	REGION 7 - Prepare output data VFD

	    REGION 7.1 - Set speed setpoint in forward and reverse direction

	        #sR_TRIG_RunFWD(CLK := #iqUDT_ConveyorInterface.RunFwd);     // Get rising edge of Run forward signal
	        #sR_TRIG_RunRVS(CLK := #iqUDT_ConveyorInterface.RunRvs);     // Get rising edge of Run reverse signal

	        // When rising edge of the forward of reverse signal is received, the drive has to stop to be able to make the switch
	        IF #sR_TRIG_RunFWD.Q OR #sR_TRIG_RunRVS.Q
	        THEN
	            #qUDT_VfdOutputs.SetpointSpeed := 0;

	        END_IF;

	        // If motor stopped and Run forward is requested and forward direction is interlock, the speed setpoint is loaded to run forward.
	        IF (#iqUDT_ConveyorInterface.RunFwd) AND #iUDT_VfdConfig.InterlockFwd //(#i_UDT_VFDInputs.ActualSpeed = 0) AND
	        THEN
	            #sx_RunVfdForward := TRUE;
	            #sx_RunVfdReverse := FALSE;
	        END_IF;

	        // If motor stopped and Run reverse is requested and reverse direction is interlock, the speed setpoint is loaded to run forward.
	        IF (#iUDT_VfdInputs.ActualSpeed = 0) AND #iqUDT_ConveyorInterface.RunRvs AND #iUDT_VfdConfig.InterlockRvs
	        THEN
	            #sx_RunVfdReverse := TRUE;
	            #sx_RunVfdForward := FALSE;
	        END_IF;

	    END_REGION

	    REGION 7.2 - Stopping

	        // Create trigger when direction signal falling
	        #sF_TRIG_RunFwd(CLK := #iqUDT_ConveyorInterface.RunFwd);
	        #sF_TRIG_RunRvs(CLK := #iqUDT_ConveyorInterface.RunRvs);

	        // When no run signal or above run signal are given or drive is running and no occurs interlock (in specific direction) the VFD should stop
	        IF (NOT #iqUDT_ConveyorInterface.RunRvs AND NOT #iqUDT_ConveyorInterface.RunFwd)
	            OR (#iqUDT_ConveyorInterface.RunRvs AND #iqUDT_ConveyorInterface.RunFwd)
	            OR (#sx_RunVfdReverse AND NOT #iUDT_VfdConfig.InterlockRvs)
	            OR (#sx_RunVfdForward AND NOT #iUDT_VfdConfig.InterlockFwd)
	            OR #sF_TRIG_RunRvs.Q
	            OR #sF_TRIG_RunFwd.Q

	        THEN
	            #sx_RunVfdReverse := FALSE;
	            #sx_RunVfdForward := FALSE;
	        END_IF;

	        IF NOT #sx_RunVfdReverse AND NOT #sx_RunVfdForward AND (#iUDT_VfdInputs.ActualSpeed <> 0)
	        THEN
	            #sx_VfdStopping := TRUE;
	        ELSE
	            #sx_VfdStopping := FALSE;
	        END_IF;

	    END_REGION

	    REGION 7.3 - Check for enable operation signal

	        #sx_EnableOperation := #sx_VfdAvailable AND NOT #sx_ConfigurationError AND (#sx_RunVfdForward OR #sx_RunVfdReverse) OR #iqUDT_ConveyorInterface.VFDRunning;

	    END_REGION

	END_REGION

	REGION 8 - Write outputs to VFD

	    REGION 8.1 - Write control word 1

	        #qUDT_VfdOutputs.Control_Word_1.EnableRapidStop := #ix_QuickStopDisable;                       // Writing state to enable VFD to run
	        #qUDT_VfdOutputs.Control_Word_1.EnableApplicationStop := #sx_EnableOperation;                  // Writing state to Enable VFD operation
	        #qUDT_VfdOutputs.Control_Word_1.ReleaseBrake := FALSE;                                         // Not used
	        #qUDT_VfdOutputs.Control_Word_1.JogPos := FALSE;                                               // Not used
	        #qUDT_VfdOutputs.Control_Word_1.JogNeg := FALSE;                                               // Not used
	        #qUDT_VfdOutputs.Control_Word_1.ApplyRelativePositioning := FALSE;                             // Not used for speed control
	        #qUDT_VfdOutputs.Control_Word_1.StartStop := #sx_EnableOperation;                              // Writing state to start or stop VFD
	        #qUDT_VfdOutputs.Control_Word_1.ResetError := #iqUDT_ConveyorInterface.InternalErrorReset;    // Reseting VFD errors with error reset bit
	        #qUDT_VfdOutputs.Control_Word_1.ActivateDriveTrain2 := FALSE;                                  // Not used for MoviGear with one Drive Train
	        #qUDT_VfdOutputs.Control_Word_1.DeactivateSW_LimitSwitch := FALSE;                             // Not used
	        #qUDT_VfdOutputs.Control_Word_1.ActivateInhibit := NOT #sx_EnableOperation;                    // Controller Inhibit has TO be "false" before start/stop
	        #qUDT_VfdOutputs.Control_Word_1.ActivateStandby := FALSE;                                      // Not used
	        #qUDT_VfdOutputs.Control_Word_1.MovikitHandshakeIn := #sx_MovikitHandshakeIn;                  // MoviKit handshake controlled BY 0.5 Hz

	        // If hardware is unavailable clear the control word
	        IF NOT #sx_VfdAvailable
	        THEN
	            #qUDT_VfdOutputs.Control_Word_1.EnableRapidStop := FALSE;                                  // Writing state to enable VFD to run
	            #qUDT_VfdOutputs.Control_Word_1.EnableApplicationStop := FALSE;                            // Writing state to Enable VFD operation
	            #qUDT_VfdOutputs.Control_Word_1.ReleaseBrake := FALSE;                                     // Not used
	            #qUDT_VfdOutputs.Control_Word_1.JogPos := FALSE;                                           // Not used
	            #qUDT_VfdOutputs.Control_Word_1.JogNeg := FALSE;                                           // Not used
	            #qUDT_VfdOutputs.Control_Word_1.ApplyRelativePositioning := FALSE;                         // NOT used FOR speed control
	            #qUDT_VfdOutputs.Control_Word_1.StartStop := FALSE;                                        // Writing state to start or stop VFD
	            #qUDT_VfdOutputs.Control_Word_1.ResetError := FALSE;                                       // Reseting VFD errors with error reset bit
	            #qUDT_VfdOutputs.Control_Word_1.ActivateDriveTrain2 := FALSE;                              // Not used for MoviGear with one Drive Train
	            #qUDT_VfdOutputs.Control_Word_1.DeactivateSW_LimitSwitch := FALSE;                         // Not used
	            #qUDT_VfdOutputs.Control_Word_1.ActivateInhibit := FALSE;                                  // Controller Inhibit has TO be "false" before start/stop
	            #qUDT_VfdOutputs.Control_Word_1.ActivateStandby := FALSE;                                  // Not used
	            #qUDT_VfdOutputs.Control_Word_1.MovikitHandshakeIn := FALSE;                               // MoviKit handshake controlled BY 0.5 Hz
	            #qUDT_VfdOutputs.Control_Word_1.BIT_02_Reserved := FALSE;
	            #qUDT_VfdOutputs.Control_Word_1.BIT_09_Reserved := FALSE;
	            #qUDT_VfdOutputs.Control_Word_1.BIT_11_Reserved := FALSE;

	        END_IF;
	    END_REGION

	    REGION 8.2 - Write speed setpoint to drive
	        // The conveyor stopped and may now run in forward direction
	        IF (#sx_RunVfdForward AND NOT #iUDT_VfdConfig.DirectionReversal)
	            OR (#sx_RunVfdReverse AND #iUDT_VfdConfig.DirectionReversal)
	        THEN
	            #qUDT_VfdOutputs.SetpointSpeed := REAL_TO_INT(#sr_ActualSpeedSetpoint);
	        END_IF;

	        // The conveyor stopped and may now run in reverse direction
	        IF (#sx_RunVfdReverse AND NOT #iUDT_VfdConfig.DirectionReversal)
	            OR (#sx_RunVfdForward AND #iUDT_VfdConfig.DirectionReversal)

	        THEN
	            #qUDT_VfdOutputs.SetpointSpeed := REAL_TO_INT(#sr_ActualSpeedSetpoint * -1);
	        END_IF;

	        // Clear speed setpoint when no run request
	        IF NOT #sx_RunVfdForward AND NOT #sx_RunVfdReverse
	        THEN
	            #qUDT_VfdOutputs.SetpointSpeed := 0;
	        END_IF;

	    END_REGION

	    REGION 8.3 - Write acceleration and deceleration value to drive
	        // Write deceleration value to VFD
	        #qUDT_VfdOutputs.SetpointAcceleration := REAL_TO_INT(#iUDT_VfdConfig.ReferenceRPM / (UDINT_TO_REAL(#iUDT_VfdConfig.VFDRampUpTime) / 1000.0));        //Recalculating Acceleration ramp - deviding maximum configured speed by Ramp up time and devide it by 1000

	        // Write deceleration value to VFD
	        #qUDT_VfdOutputs.SetpointDeceleration := REAL_TO_INT(#iUDT_VfdConfig.ReferenceRPM / (UDINT_TO_REAL(#iUDT_VfdConfig.VFDRampDownTime) / 1000.0));      //Recalculating Deceleration ramp - deviding maximum configured speed by Ramp down time and devide it by 1000

	    END_REGION

	END_REGION

	REGION 9 - Check if motor is running

	    //The moto should start running after specific time. If nit the VFDRunningFeedback error occured
	    #sFB_TimerOnOffDelayVFDRunningFeedbackError(iudi_OnDelayTime := #iUDT_VfdConfig.VFDStartupTime,
	                                                ix_SignalToDelay := #sx_EnableOperation AND NOT (#si_ActualSpeed <> 0));

	    IF #sFB_TimerOnOffDelayVFDRunningFeedbackError.qx_DelayedSignal THEN

	        #sUDT_HMIStatus.VFDRunningFeedbackError := TRUE;

	    END_IF;

	END_REGION

	REGION 10 - Copy signals to interface DB and to status output UDT
	    // Create internal error status
	    #sx_ErrorActive := #sUDT_HMIStatus.PNSlaveNotonline
	    OR #sUDT_HMIStatus.PNSlaveError
	    OR #sUDT_HMIStatus.InternalError
	    OR #sUDT_HMIStatus.CommunicationErrorMovikit
	    OR #sUDT_HMIStatus.VFDRunningFeedbackError;

	    // Write interface bits
	    #iqUDT_ConveyorInterface.VFDRunning := #iUDT_VfdInputs.Status_Word_1.DriveActive AND #sx_VfdAvailable AND #iqUDT_ConveyorInterface.ActualSpeed <> 0;        // Write true on output Conveyor interface structure if VFD is in operation and motor is turning
	    #iqUDT_ConveyorInterface.VFDatSpeed := #sx_SpeedSetpointReached AND #sx_VfdAvailable;                                                                         // Copy setpoint speed reached state from static  to the output conveyor interface structure
	    #iqUDT_ConveyorInterface.InternalWarningVFD := #iUDT_VfdInputs.Status_Word_1.Warning;                                                                         // Set the internal VFD warning bit if any warning is active
	    #iqUDT_ConveyorInterface.InternalErrorVFD := #sx_ErrorActive;                                                                                                  // Set the internal VFD error bit if any fault is active
	    #iqUDT_ConveyorInterface.ActualSpeed := #si_ActualSpeed;                                                                                                       // Copy the calculated value to the output
	    #iqUDT_ConveyorInterface.ConfigurationError := #iqUDT_ConveyorInterface.ConfigurationError OR #sx_ConfigurationError;

	    // Copy error status to output
	    #qUDT_HMIStatus := #sUDT_HMIStatus;
	END_REGION

	REGION 11 - Statistics
	    // Create trigger on error and create statistics for profinet slave not online
	    #sR_TRIG_PNSlaveNotOnline(CLK := #sUDT_HMIStatus.PNSlaveNotonline);                              // Detect the rising edge of the error

	    IF #iqUDT_ConveyorInterface.ResetStatistics OR #sUDT_HMIStatus.PNSlaveNotonline
	    THEN

	        "FC_Statistics"(ix_Reset := #iqUDT_ConveyorInterface.ResetStatistics,
	                        ix_Activate := #sUDT_HMIStatus.PNSlaveNotonline,
	                        ix_RTrigActivate := #sR_TRIG_PNSlaveNotOnline.Q,
	                        iqUDT_Statistics := #iqUDT_VfdStatistics.PNSlaveNotOnline);
	    END_IF;

	    // Create trigger on error and create statistics for profinet slave error
	    #sR_TRIG_PNSlaveError(CLK := #sUDT_HMIStatus.PNSlaveError);                                      // Detect the rising edge of the error

	    IF #iqUDT_ConveyorInterface.ResetStatistics OR #sUDT_HMIStatus.PNSlaveError
	    THEN

	        "FC_Statistics"(ix_Reset := #iqUDT_ConveyorInterface.ResetStatistics,
	                        ix_Activate := #sUDT_HMIStatus.PNSlaveError,
	                        ix_RTrigActivate := #sR_TRIG_PNSlaveError.Q,
	                        iqUDT_Statistics := #iqUDT_VfdStatistics.PNSlaveError);
	    END_IF;

	    // Create trigger on error and create statistics for internal VFD Error
	    #sR_TRIG_InternalError(CLK := #sUDT_HMIStatus.InternalError);                                    // Detect the rising edge of the error

	    IF #iqUDT_ConveyorInterface.ResetStatistics OR #sUDT_HMIStatus.InternalError
	    THEN

	        "FC_Statistics"(ix_Reset := #iqUDT_ConveyorInterface.ResetStatistics,
	                        ix_Activate := #sUDT_HMIStatus.InternalError,
	                        ix_RTrigActivate := #sR_TRIG_InternalError.Q,
	                        iqUDT_Statistics := #iqUDT_VfdStatistics.VFDInternalError);
	    END_IF;

	    // Create trigger on error and create statistics for Movikit communication error
	    #sR_TRIG_CommunicationErrorMovikit(CLK := #sUDT_HMIStatus.CommunicationErrorMovikit);            // Detect the rising edge of the error

	    IF #iqUDT_ConveyorInterface.ResetStatistics OR #sUDT_HMIStatus.CommunicationErrorMovikit
	    THEN

	        "FC_Statistics"(ix_Reset := #iqUDT_ConveyorInterface.ResetStatistics,
	                        ix_Activate := #sUDT_HMIStatus.CommunicationErrorMovikit,
	                        ix_RTrigActivate := #sR_TRIG_CommunicationErrorMovikit.Q,
	                        iqUDT_Statistics := #iqUDT_VfdStatistics.CommunicationErrorMovikit);
	    END_IF;

	    // Create trigger on running signal and create statistics for running status
	    #sR_TRIG_Running(CLK := #iqUDT_ConveyorInterface.VFDRunning);                                 // Detect the rising edge of the signal

	    IF #iqUDT_ConveyorInterface.ResetStatistics OR #iqUDT_ConveyorInterface.VFDRunning
	    THEN

	        "FC_Statistics"(ix_Reset := #iqUDT_ConveyorInterface.ResetStatistics,
	                        ix_Activate := #iqUDT_ConveyorInterface.VFDRunning,
	                        ix_RTrigActivate := #sR_TRIG_Running.Q,
	                        iqUDT_Statistics := #iqUDT_VfdStatistics.Running);
	    END_IF;
	END_REGION

	REGION 12 - VFD codes
	    (*
	    FCB number |                       | Meaning
	    ______________________________________________________________________________________________________________
	        1                               Output stage inhibit
	        2                               Default stop
	        4                               Manual Mode
	        5                               Speed control
	                101                     Speed-controlled jogging. Encoder feedback NOT required.
	                200                     Speed control. Encoder feedback NOT required.
	        6                               Interpolated speed control
	        7                               Torque control
	        8                               Interpolated torque control
	        9                               Positioning mode
	                400                     Absolute position control
	                401                     Relative position control
	                402                     Modulo position control - positive
	                403                     Modulo position control - negative
	                404                     Modulo position control - shortest distance
	        10                              Interpolated position control
	        12                              Referencing mode
	                300                     Reference travel - offset via parameter
	                301                     Reference travel - offset via fieldbus
	        13                              Stop at application limits
	        14                              Emergency stop
	        18                              Rotor position identification
	        19                              Position hold control
	        20                              Jog mode
	                100                     Position-controlled jogging. Encoder feedback required
	        21                              Brake test
	        25                              Motor parameter measurement
	        26                              Stop at user limits

	    Error code | Suberror code        | Meaning                                | Measure
	    ______________________________________________________________________________________________________________
	        3       1                       Ground fault                            Consult "Fault table" in
	        4       1                       Brake chopper fault                     document 'SEW Movigear-C 25887130.PDF'
	        6       1                       Line fault                              Chapter 8.7
	        7       1                       DC link fault
	        8       1,2,3                   Speed monitoring fault
	        9       1,2,5,6,9,10            Control mode fault
	        10      1,3-11                  Data flexibility fault
	        11      1-6                     Temperature monitoring fault
	        12      1,2                     Fault brake
	        13      5,24                    Encoder 1 fault
	        16      5-8,10,20-27            Startup fault
	        19      1-9                     Process data fault
	        20      2,11                    Fault device monitoring
	        23      4                       Power section fault
	        25      2-7,20,21,30,31,61,70   Parameter memory monitoring
	        26      1,3                     External fault
	        28      1-12,14                 FCB drive function fault
	        29      1-4                     Hardware limit switch fault
	        30      1-3                     Software limit switch fault
	        31      1-4,7,9                 Thermal protection fault
	        32      2-6,12                  Communication fault
	        33      11,12,13                system initialisation fault
	        34      1                       Process data configuration fault
	        35      1-5                     Function activation fault
	        42      1-3                     Lag fault
	        46      2,3,50,51,52            Safety card fault
	        51      1                       Analog processing fault

	    Error code | Suberror code        | Meaning                                | Measure
	    ______________________________________________________________________________________________________________
	        1       1,2                     Output stage monitoring fault           Contact SEW-Eurodrive Service
	        4       2                       Brake chopper fault
	        7       2                       DC link fault
	        9       3,4,8                   Control mode fault
	        10      2,99                    Data flexibility fault
	        11      7,8                     Temperature monitoring fault
	        13      1,3,6,7.8,9,11,13,      Encoder 1 fault
	                15,22,23
	        16      2,11,12,30              Startup fault
	        17      7                       Internal processor fault
	        18      1,3,4,7,8,9,10,12,13    Software fault
	        20      1,7                     Fault device monitoring
	        21      1                       S-Drive 1 fault
	        23      5,6,7,8                 Power section fault
	        25      10,12-19,50,51,81       Parameter memory monitoring
	        28      13                      FCB drive funcyio fault
	        33      1,2,6,7,8,10            System initialisation fault
	        46      1                       Safety card fault

	    Function Control Block (FCB) codes
	    FBC = 01 Output stage inhibit
	    FBC = 02 Default stop
	    FBC = 04 Manual Mode
	    FBC = 05 Speed control
	     101 - Speed-controlled jogging. Encoder feedback NOT required.
	     200 - Speed control. Encoder feedback NOT required.
	    FBC = 06 Interpolated speed control
	    FBC = 07 Torque control
	    FBC = 08 Interpolated torque control
	    FBC = 09 Positioning mode
	    400 - Absolute position control
	    401 - Relative position control
	    402 - Modulo position control - positive
	    403 - Modulo position control - negative
	    404 - Modulo position control - shortest distance
	    FBC = 10 Interpolated position control
	    FBC = 12 Referencing mode
	    300 - Reference travel - offset via parameter
	    301 - Reference travel - offset via fieldbus
	    FBC = 13 Stop at application limits
	    FBC = 14 Emergency stop
	    FBC = 18 Rotor position identification
	    FBC = 19 Position hold control
	    FBC = 20 Jog mode
	     100 - Position-controlled jogging. Encoder feedback required
	    FBC = 21 Brake test
	    FBC = 25 Motor parameter measurement
	    FBC = 26 Stop at user limits

	    *)
	END_REGION
END_FUNCTION_BLOCK

FUNCTION_BLOCK "FB_VfdSEWMOVI-CPositioning"
TITLE = FB_VFD_SEW_MOVI-C_Positioning
{ S7_Optimized_Access := 'TRUE' }
AUTHOR : MHSE
VERSION : 3.0
// ATTRIBUTES
// AUTO_NUMBER = True
// BLOCK_NUMBER = 36
// END_ATTRIBUTES
//Control SEW Servo VFD with multiple positions
   VAR_INPUT
      iUDT_VfdConfig { ExternalAccessible := 'False'; ExternalVisible := 'False'; ExternalWritable := 'False'} : "UDT_VfdPositioningConfiguration";   //  Configuration structure
      iUDT_VfdInputs { ExternalAccessible := 'False'; ExternalVisible := 'False'; ExternalWritable := 'False'} : "UDT_VfdSEWPositioningPI";   //  VFD inputs structure
      ix_MainPowerOk { ExternalAccessible := 'False'; ExternalVisible := 'False'; ExternalWritable := 'False'} : Bool;   //  True = Main power is ok
      ix_BackupPowerOk { ExternalAccessible := 'False'; ExternalVisible := 'False'; ExternalWritable := 'False'} : Bool;   //  True = back-up power is ok
      ix_SimulationModeActive { ExternalAccessible := 'False'; ExternalVisible := 'False'; ExternalWritable := 'False'} : Bool;   //  Simulation On
   END_VAR

   VAR_OUTPUT
      qUDT_HMIStatus { ExternalAccessible := 'False'; ExternalVisible := 'False'; ExternalWritable := 'False'} : "UDT_VfdPositioningStatus";   //  HMI status structure
      qUDT_VfdOutputs { ExternalAccessible := 'False'; ExternalVisible := 'False'; ExternalWritable := 'False'} : "UDT_VfdSEWPositioningPO";   //  VFD outputs structure
   END_VAR

   VAR_IN_OUT
      iqUDT_VSUInterface : "UDT_VSUInterface";   //  VSU interface structure
      iqUDT_VFDStatistics : "UDT_VfdStatistics";   //  VFD statistics
   END_VAR

   VAR
      sUDT_PNDevice { ExternalAccessible := 'False'; ExternalVisible := 'False'; ExternalWritable := 'False'; S7_SetPoint := 'False'} : "UDT_PNDevice";   //  PN device info structure
      sUDT_HMIStatus { ExternalAccessible := 'False'; ExternalVisible := 'False'; ExternalWritable := 'False'; S7_SetPoint := 'False'} : "UDT_VfdPositioningStatus";   //  Status struture
      sFB_TimerOnOffDelayCheckSupply { ExternalAccessible := 'False'; ExternalVisible := 'False'; ExternalWritable := 'False'; S7_SetPoint := 'False'} : "FB_TimerOnOffDelay";   //  MHS "TimerOnOffDelay" - to delay time for VFD supply contactor
      sFB_TimerOnOffDelayMoviKit { ExternalAccessible := 'False'; ExternalVisible := 'False'; ExternalWritable := 'False'; S7_SetPoint := 'False'} : "FB_TimerOnOffDelay";   //  MHS "TimerOnOffDelay" - to delay time for MoviKit response delay error
      sFB_TimerOnOffDelayPositioning { ExternalAccessible := 'False'; ExternalVisible := 'False'; ExternalWritable := 'False'; S7_SetPoint := 'False'} : "FB_TimerOnOffDelay";   //  MHS "TimerOnOffDelay" - to delay time for Porisioning delay error
      sFB_TimerOnOffDelayFasterManualSpeed { ExternalAccessible := 'False'; ExternalVisible := 'False'; ExternalWritable := 'False'; S7_SetPoint := 'False'} : "FB_TimerOnOffDelay";
      sFB_TimerOnOffDelayActivateInhibit { ExternalAccessible := 'False'; ExternalVisible := 'False'; ExternalWritable := 'False'; S7_SetPoint := 'False'} : "FB_TimerOnOffDelay";
      sF_TRIG_LST {InstructionName := 'F_TRIG'; LibVersion := '1.0'; ExternalAccessible := 'False'; ExternalVisible := 'False'; ExternalWritable := 'False'; S7_SetPoint := 'False'} : F_TRIG;   //  Falling edge positioning feedback
      sR_TRIG_ManInPos {InstructionName := 'R_TRIG'; LibVersion := '1.0'; ExternalAccessible := 'False'; ExternalVisible := 'False'; ExternalWritable := 'False'; S7_SetPoint := 'False'} : R_TRIG;   //  Rising edge manual travel into position
      sR_TRIG_PNSlaveNotOnline {InstructionName := 'R_TRIG'; LibVersion := '1.0'; ExternalAccessible := 'False'; ExternalVisible := 'False'; ExternalWritable := 'False'; S7_SetPoint := 'False'} : R_TRIG;   //  Rising edge for trigger Profinet slave not online statistics
      sR_TRIG_PNSlaveError {InstructionName := 'R_TRIG'; LibVersion := '1.0'; ExternalAccessible := 'False'; ExternalVisible := 'False'; ExternalWritable := 'False'; S7_SetPoint := 'False'} : R_TRIG;   //  Rising edge for trigger Profinet slave error statistics
      sR_TRIG_InternalError {InstructionName := 'R_TRIG'; LibVersion := '1.0'; ExternalAccessible := 'False'; ExternalVisible := 'False'; ExternalWritable := 'False'; S7_SetPoint := 'False'} : R_TRIG;   //  Rising edge for trigger Internal VFD Error statistics
      sR_TRIG_CommunicationErrorMovikit {InstructionName := 'R_TRIG'; LibVersion := '1.0'; ExternalAccessible := 'False'; ExternalVisible := 'False'; ExternalWritable := 'False'; S7_SetPoint := 'False'} : R_TRIG;   //  Rising edge for trigger communication error Movikit statistics
      sR_TRIG_Running {InstructionName := 'R_TRIG'; LibVersion := '1.0'; ExternalAccessible := 'False'; ExternalVisible := 'False'; ExternalWritable := 'False'; S7_SetPoint := 'False'} : R_TRIG;   //  Rising edge for starting of the running signal
      sa_PNPortsStatus { ExternalAccessible := 'False'; ExternalVisible := 'False'; ExternalWritable := 'False'} : Array[1..8] of Bool;   // TRUE when specific port has an error
      sr_ActualTorque { ExternalAccessible := 'False'; ExternalVisible := 'False'; ExternalWritable := 'False'} : Real;   //  Actual torque of drive
      sdi_ActualPositionValue { ExternalAccessible := 'False'; ExternalVisible := 'False'; ExternalWritable := 'False'} : DInt;   //  Actual position in mm
      si_ManualSpeed { ExternalAccessible := 'False'; ExternalVisible := 'False'; ExternalWritable := 'False'} : Int;   //  Actual manual speed
      si_ActualSpeed { ExternalAccessible := 'False'; ExternalVisible := 'False'; ExternalWritable := 'False'} : Int;   //  Actual speed in mm/s
      si_LastSwitchtime { ExternalAccessible := 'False'; ExternalVisible := 'False'; ExternalWritable := 'False'} : Int;   //  The actual time it took the last switch-over
      sx_ErrorActive { ExternalAccessible := 'False'; ExternalVisible := 'False'; ExternalWritable := 'False'} : Bool;   //  An error is active
      sx_WarningActive { ExternalAccessible := 'False'; ExternalVisible := 'False'; ExternalWritable := 'False'} : Bool;   //  A warning is active
      sx_PNDeviceHealthy { ExternalAccessible := 'False'; ExternalVisible := 'False'; ExternalWritable := 'False'} : Bool;   //  PN Device is healthy, no errors
      sx_MovikitHandshakeIn { ExternalAccessible := 'False'; ExternalVisible := 'False'; ExternalWritable := 'False'} : Bool;   //  Handshake to movikit
      sx_MoviKitFeedback { ExternalAccessible := 'False'; ExternalVisible := 'False'; ExternalWritable := 'False'} : Bool;   //  Movikit feedback delay
      sx_HardwareAvailable { ExternalAccessible := 'False'; ExternalVisible := 'False'; ExternalWritable := 'False'} : Bool;   //  All hardware is on line and available
      sx_PowerOK { ExternalAccessible := 'False'; ExternalVisible := 'False'; ExternalWritable := 'False'} : Bool;   //  All Power (in and external) is ok
      sx_PositioningFeedback { ExternalAccessible := 'False'; ExternalVisible := 'False'; ExternalWritable := 'False'} : Bool;   //  Positioning feedback delay
      sx_VFDReady { ExternalAccessible := 'False'; ExternalVisible := 'False'; ExternalWritable := 'False'} : Bool;   //  The VFD control is ready to operate
      sx_StartVFD { ExternalAccessible := 'False'; ExternalVisible := 'False'; ExternalWritable := 'False'} : Bool;   //  Start VFD
      sx_MotorRunning { ExternalAccessible := 'False'; ExternalVisible := 'False'; ExternalWritable := 'False'} : Bool;   //  The servo motor is running
      sx_ManualPositionStop { ExternalAccessible := 'False'; ExternalVisible := 'False'; ExternalWritable := 'False'} : Bool;   //  A configured position is reached in manual mode
      sx_ManualPosHold { ExternalAccessible := 'False'; ExternalVisible := 'False'; ExternalWritable := 'False'} : Bool;   //  Hold in position
      sx_RestartMan { ExternalAccessible := 'False'; ExternalVisible := 'False'; ExternalWritable := 'False'} : Bool;   //  Manual restart requested
      sx_ConfigurationError { ExternalAccessible := 'False'; ExternalVisible := 'False'; ExternalWritable := 'False'} : Bool;   //  Commissioning: configuration of parameters is wrong
      si_LoopCounter { ExternalAccessible := 'False'; ExternalVisible := 'False'; ExternalWritable := 'False'} : Int;
      sx_Check { ExternalAccessible := 'False'; ExternalVisible := 'False'; ExternalWritable := 'False'} : Bool;
   END_VAR

   VAR_TEMP
      tdi_EncoderPositionSetpoint : DInt;   //  Value of position setpoint
   END_VAR

   VAR CONSTANT
      ci_NumberOfProfinetPorts : Int := 2;   // Number of Profinet ports in device
      ci_SpeedManualMode : Int := 100;   // Speed in manual mode for jogging
      ci_SpeedManualModeAfter5s : Int := 200;
   END_VAR


BEGIN
	(*
	----------------------------------------------------------------------------------------

	Version history:
	Date        | Version   | Author        | Remark
	----------------------------------------------------------------------------------------
	24/05/2019  | 0.1       | P. Majka      | first release MHS TIA 15.1
	29/07/2019  | 0.2       | P. Majka      | Adding new functionality - comments to change
	30/07/2019  | 2.0       | P. Majka      | Moved to project with library 2.0
	31/07/2019  | 2.1       | M. Kurpiers   | Updating comments
	08/08/2019  | 2.2       | J.Krawczuk    | Updating referencing
	14/08/2019  | 2.3       | J.Krawczuk    | Added new functionality
	24/08/2019  | 2.4       | F. Baten      | Changed regions / combined errors / modified comments and working
	05/11/2019  | 2.5       | S.Theocharis  | Change the VFDDeviceName to VFDPNDeviceName for consistency with rest VFD blocks
	20/11/2019  | 2.10      | S. Nikodem    | Configuration error
	20/11/2019  | 3.0       | P.Majka       | 3.0 MHS library release TIA 15.1
	28/02/2020  | 3.1       | F.Baten       | Reinstated positioning warning (Servo takes too long to get to position) and
	                                        | separated it again from OutOfPosition error (over running the set positions)
	01/02/2020  | 3.2       | F.Baten       | Changed "UDT_VFD_Status" to "UDT_VFD_PositioningStatus"
	04/02/2020  | 3.3       | F.Baten       | Changed VSU Rio interface - Error and ready modified.
	06/08/2020  | 3.4       | L.Klar        | Manual speed changed
	03/11/2020  | 3.5       | K.Pokorski    | Profinet ports diagnostics added
	21/02/2023  | 4.0       | F.Baten       | 4.0 Release TIA 17.5
	06/10/2023  | 4.1       | F.Baten       | All positions converted to DINT as need of higher values for lift funtion
	14/06/2024  | 4.1       | R.Pieczonka   | Changed conditions for "EnableApplicationStop". Fixed setting output speed
	*)

	REGION 1 - Get Device Profinet information

	    "FC_GetDevicePN"(is_PNDeviceName := #iUDT_VfdConfig.VFDPNDeviceName,
	                     ix_SimulationModeActive := #ix_SimulationModeActive,
	                     iqUDT_PND := #sUDT_PNDevice);


	    "FC_GetPNPortStatus"(ii_NumberOfPorts := #ci_NumberOfProfinetPorts,
	                         iUDT_DevicePNInfo := #sUDT_PNDevice,
	                         qa_PortFault => #sa_PNPortsStatus);

	END_REGION

	REGION 2 - Reset errors

	    IF #iqUDT_VSUInterface.InternalErrorReset

	    THEN
	        #sUDT_HMIStatus.CommunicationErrorMovikit := FALSE;                    // The Movikit application is not reacting
	        #sUDT_HMIStatus.PNSlaveNotOnline := FALSE;                             // Profinet slave is not on line
	        #sUDT_HMIStatus.PNSlaveError := FALSE;                                 // Profinet slave has an error
	        #sUDT_HMIStatus.PositioningTimeOutError := FALSE;                      // Reset positioning error
	        #sUDT_HMIStatus.InternalError := FALSE;                                // Reset internal error
	        #sUDT_HMIStatus.PNSlaveWarning := FALSE;


	    END_IF;

	END_REGION

	REGION 3 - Check Hardware

	    REGION 3.1 - Power OK
	        // Hardware will be available after delay so the device has time for initialisation
	        #sFB_TimerOnOffDelayCheckSupply(iudi_OnDelayTime := 2000,              // Set time for on delay
	                                        ix_SignalToDelay := #ix_MainPowerOk);  // Mains are ok

	        #sx_PowerOK := #sFB_TimerOnOffDelayCheckSupply.qx_DelayedSignal;       // And All Power (in and external) is ok
	    END_REGION

	    REGION 3.2 - PN Healthy Check

	        IF NOT "DB_ProfinetDiagnostic".ProfinetNetworks[#sUDT_PNDevice.PNNetworknumber].DeviceStatus[#sUDT_PNDevice.PNDeviceNumber].DeviceState.Exist     // Or the connected device doesn't exist
	            AND NOT #ix_SimulationModeActive                                    // And not in simulation
	            AND (#sx_PowerOK                                                    // Main Power is ok
	            OR #ix_BackupPowerOk)                                               // Or backup power is ok
	        THEN
	            #sUDT_HMIStatus.PNSlaveNotOnline := TRUE;
	        END_IF;

	        // Check if PN ports are healthy
	        IF #sa_PNPortsStatus[1] XOR #sa_PNPortsStatus[2] THEN
	            #sUDT_HMIStatus.PNSlaveWarning := TRUE;
	        END_IF;

	        IF "DB_ProfinetDiagnostic".ProfinetNetworks[#sUDT_PNDevice.PNNetworknumber].DeviceStatus[#sUDT_PNDevice.PNDeviceNumber].DeviceState.Error       // Or the device has an error
	            AND NOT #ix_SimulationModeActive                                    // And not in simulation
	            AND (#sx_PowerOK                                                    // Main Power is ok
	            OR #ix_BackupPowerOk)                                               // Or backup power is ok
	            AND NOT #sUDT_HMIStatus.PNSlaveWarning                             // and PN ports are healthy

	        THEN
	            #sUDT_HMIStatus.PNSlaveError := TRUE;                              // Profinet slave has an error
	        END_IF;

	        #sx_PNDeviceHealthy := NOT #sUDT_HMIStatus.PNSlaveNotOnline            // Or the device an error
	        AND NOT #sUDT_HMIStatus.PNSlaveError                                   // Profinet slave has an error
	        AND (#sx_PowerOK                                                        // Main Power is ok
	        OR #ix_BackupPowerOk)                                                   // Or backup power is ok
	        AND #sUDT_PNDevice.PNDeviceFound;                                      // Device is found in network configuration

	    END_REGION

	    // Hardware is available
	    #sx_HardwareAvailable := #iUDT_VfdInputs.Status_Word_1.STO_Inactive        // Safety is ok
	    AND #sx_PowerOK                                                             // All mains are ok
	    AND #sx_PNDeviceHealthy                                                     // No PN errors
	    OR #ix_SimulationModeActive;                                                // Or simulation active

	    REGION 3.3 - Check communication MoviKit
	        #sx_MoviKitFeedback :=                                                  // Set MoviKit feedback delay
	        ((#sx_MovikitHandshakeIn                                                // IF MoviKit handshake input is active
	        AND NOT #iUDT_VfdInputs.Status_Word_1.MovikitHandshakeOut)             // And MoviKit handshake output active
	        OR (NOT #sx_MovikitHandshakeIn                                          // Or MoviKit handshake input isn't active
	        AND #iUDT_VfdInputs.Status_Word_1.MovikitHandshakeOut));               // And MoviKit handshake output isn't active

	        #sFB_TimerOnOffDelayMoviKit(iudi_OnDelayTime := 1000,                  // Set on delay time to 1000
	                                    ix_SignalToDelay := NOT #sx_MoviKitFeedback);          // Start timer

	        IF (#sFB_TimerOnOffDelayMoviKit.qx_DelayedSignal)                      // If the timer elapsed
	            AND #sx_HardwareAvailable
	        THEN
	            #sUDT_HMIStatus.CommunicationErrorMovikit := TRUE;                 // Set MoviKit error
	        END_IF;

	        #sx_MovikitHandshakeIn := NOT #iUDT_VfdInputs.Status_Word_1.MovikitHandshakeOut;   // Set the Handshake signal
	    END_REGION


	END_REGION

	REGION 4 - Handle input data

	    REGION 4.1 - Move to status

	        #sr_ActualTorque := INT_TO_REAL(#iUDT_VfdInputs.ActualTorque) / 1000.0 * #iUDT_VfdConfig.TorqueMax;   // Writing actual real calculated torque
	        #si_ActualSpeed := #iUDT_VfdInputs.ActualSpeed;                                                        // Actual speed in mm/s
	        #sx_MotorRunning := #iUDT_VfdInputs.Status_Word_1.DriveActive;                                         // Set status motor running if motor shaft is turning

	    END_REGION

	    REGION 4.2 - Actual positon value

	        #sdi_ActualPositionValue := SHL(IN := (WORD_TO_DINT(IN := #iUDT_VfdInputs.ActualPosition_hW)), N := 16) + WORD_TO_DINT(IN := #iUDT_VfdInputs.ActualPosition_lW);   // Calculate actual encoder position from two words

	        IF #sdi_ActualPositionValue <= (#iUDT_VfdConfig.Position[#iqUDT_VSUInterface.PositionSetpoint] + #iUDT_VfdConfig.PositionWindow)         // If actual encoder position in mm is lower or equal to position setpoint plus position window
	            AND #sdi_ActualPositionValue >= (#iUDT_VfdConfig.Position[#iqUDT_VSUInterface.PositionSetpoint] - #iUDT_VfdConfig.PositionWindow)    // And actual encoder position in mm is greater or equal to position setpoint minus position window

	        THEN
	            #iqUDT_VSUInterface.PositionActual := #iqUDT_VSUInterface.PositionSetpoint;                                              // Write position setpoint TO actual position number when position setpoint reached
	        ELSIF #iqUDT_VSUInterface.Manual
	        THEN
	            #sx_Check := FALSE;
	            FOR #si_LoopCounter := 0 TO "FC_GetNrOfArrayEl"(iv_Array := #iUDT_VfdConfig.Position) DO
	                IF #sdi_ActualPositionValue <= (#iUDT_VfdConfig.Position[#si_LoopCounter] + #iUDT_VfdConfig.PositionWindow)
	                    AND #sdi_ActualPositionValue >= (#iUDT_VfdConfig.Position[#si_LoopCounter] - #iUDT_VfdConfig.PositionWindow)
	                THEN
	                    #iqUDT_VSUInterface.PositionActual := #si_LoopCounter;
	                    #sx_Check := TRUE;
	                END_IF;
	            END_FOR;
	            IF #sx_Check = 0 THEN
	                #iqUDT_VSUInterface.PositionActual := 0;
	            END_IF;
	        ELSE
	            #iqUDT_VSUInterface.PositionActual := 0;
	        END_IF;




	    END_REGION

	    REGION 4.3 - Manual position
	        // to stop at a predefined position when jogging, after the stop the movement can continue by pressing the jogbutton again
	        IF #iUDT_VfdInputs.Mode = 100                                                                          // The actual application mode is equal to 100
	        THEN
	            #sx_ManualPositionStop :=
	            (#sdi_ActualPositionValue <= (#iUDT_VfdConfig.Position[1] + #iUDT_VfdConfig.PositionWindow)       // IF actual encoder position in mm is lower OR equal TO position setpoint plus position window
	            AND #sdi_ActualPositionValue >= (#iUDT_VfdConfig.Position[1] - #iUDT_VfdConfig.PositionWindow))   // And actual encoder position in mm is greater or equal to position setpoint minus position window
	            OR (#sdi_ActualPositionValue <= (#iUDT_VfdConfig.Position[2] + #iUDT_VfdConfig.PositionWindow)    // IF actual encoder position in mm is lower OR equal TO position setpoint plus position window
	            AND #sdi_ActualPositionValue >= (#iUDT_VfdConfig.Position[2] - #iUDT_VfdConfig.PositionWindow))   // And actual encoder position in mm is greater or equal to position setpoint minus position window
	            OR (#sdi_ActualPositionValue <= (#iUDT_VfdConfig.Position[3] + #iUDT_VfdConfig.PositionWindow)    // IF actual encoder position in mm is lower OR equal TO position setpoint plus position window
	            AND #sdi_ActualPositionValue >= (#iUDT_VfdConfig.Position[3] - #iUDT_VfdConfig.PositionWindow))   // And actual encoder position in mm is greater or equal to position setpoint minus position window
	            OR (#sdi_ActualPositionValue <= (#iUDT_VfdConfig.Position[4] + #iUDT_VfdConfig.PositionWindow)    // IF actual encoder position in mm is lower OR equal TO position setpoint plus position window
	            AND #sdi_ActualPositionValue >= (#iUDT_VfdConfig.Position[4] - #iUDT_VfdConfig.PositionWindow))   // And actual encoder position in mm is greater or equal to position setpoint minus position window
	            OR (#sdi_ActualPositionValue <= (#iUDT_VfdConfig.Position[5] + #iUDT_VfdConfig.PositionWindow)    // IF actual encoder position in mm is lower OR equal TO position setpoint plus position window
	            AND #sdi_ActualPositionValue >= (#iUDT_VfdConfig.Position[5] - #iUDT_VfdConfig.PositionWindow))   // And actual encoder position in mm is greater or equal to position setpoint minus position window
	            OR (#sdi_ActualPositionValue <= (#iUDT_VfdConfig.Position[6] + #iUDT_VfdConfig.PositionWindow)    // IF actual encoder position in mm is lower OR equal TO position setpoint plus position window
	            AND #sdi_ActualPositionValue >= (#iUDT_VfdConfig.Position[6] - #iUDT_VfdConfig.PositionWindow))   // And actual encoder position in mm is greater or equal to position setpoint minus position window
	            OR (#sdi_ActualPositionValue <= (#iUDT_VfdConfig.Position[7] + #iUDT_VfdConfig.PositionWindow)    // IF actual encoder position in mm is lower OR equal TO position setpoint plus position window
	            AND #sdi_ActualPositionValue >= (#iUDT_VfdConfig.Position[7] - #iUDT_VfdConfig.PositionWindow))   // And actual encoder position in mm is greater or equal to position setpoint minus position window
	            OR (#sdi_ActualPositionValue <= (#iUDT_VfdConfig.Position[8] + #iUDT_VfdConfig.PositionWindow)    // IF actual encoder position in mm is lower OR equal TO position setpoint plus position window
	            AND #sdi_ActualPositionValue >= (#iUDT_VfdConfig.Position[8] - #iUDT_VfdConfig.PositionWindow))   // And actual encoder position in mm is greater or equal to position setpoint minus position window
	            OR (#sdi_ActualPositionValue <= (#iUDT_VfdConfig.Position[9] + #iUDT_VfdConfig.PositionWindow)    // IF actual encoder position in mm is lower OR equal TO position setpoint plus position window
	            AND #sdi_ActualPositionValue >= (#iUDT_VfdConfig.Position[9] - #iUDT_VfdConfig.PositionWindow))   // And actual encoder position in mm is greater or equal to position setpoint minus position window
	            OR (#sdi_ActualPositionValue <= (#iUDT_VfdConfig.Position[10] + #iUDT_VfdConfig.PositionWindow)   // IF actual encoder position in mm is lower OR equal TO position setpoint plus position window
	            AND #sdi_ActualPositionValue >= (#iUDT_VfdConfig.Position[10] - #iUDT_VfdConfig.PositionWindow)); // And actual encoder position in mm is greater or equal to position setpoint minus position window
	        END_IF;
	    END_REGION
	END_REGION

	REGION 5 - Errors and warnings

	    REGION 5.1 - VFD internal error

	        #sUDT_HMIStatus.InternalError := #iUDT_VfdInputs.Status_Word_1.Error; // An internal VFD error is active
	        #sUDT_HMIStatus.ErrorCode := #iUDT_VfdInputs.StatusErrorNo.%B1;       // Copy VFD error code from static status structure to HMI status structure
	        #sUDT_HMIStatus.SubErrorCode := #iUDT_VfdInputs.StatusErrorNo.%B0;    // Copy VFD sub-error code from static status structure to HMI status structure

	        IF NOT #iUDT_VfdInputs.Status_Word_1.Error
	            AND NOT #iUDT_VfdInputs.Status_Word_1.Warning
	        THEN
	            #sUDT_HMIStatus.ErrorCode := 0;                                    // Copy VFD error code from static status structure TO HMI status structure
	            #sUDT_HMIStatus.SubErrorCode := 0;                                 // Copy VFD sub-error code from static status structure to HMI status structure
	        END_IF;
	    END_REGION

	    REGION 5.2 - Positioning error
	        // This timer checks if the speed of the VFD is ok.
	        // The VFD should reach is next destination in the given time
	        //

	        #sx_PositioningFeedback := #iqUDT_VSUInterface.PositionActual <> #iqUDT_VSUInterface.PositionSetpoint // If actual position is different than setpoint position
	        AND #iqUDT_VSUInterface.Automatic;                                                                     // And in automatic mode

	        #sF_TRIG_LST(CLK := #sx_PositioningFeedback);

	        IF #sF_TRIG_LST.Q
	        THEN
	            #si_LastSwitchtime := LREAL_TO_INT(#sFB_TimerOnOffDelayPositioning.qlr_ActualTime);
	        END_IF;



	        #sFB_TimerOnOffDelayPositioning(iudi_OnDelayTime := (#iqUDT_VSUInterface.SwitchingTime),  // Set on delay time
	                                        ix_SignalToDelay := #sx_PositioningFeedback);              // Start timer when positioning feedback delay



	        IF #sFB_TimerOnOffDelayPositioning.qx_DelayedSignal                    // If the time elapsed
	        THEN

	            #sUDT_HMIStatus.PositioningTimeOutError := TRUE;                   // Set positioning warning

	        END_IF;
	    END_REGION

	    REGION 5.3 - Common Error
	        // Set VFD error active
	        #sx_ErrorActive := #sUDT_HMIStatus.InternalError                       // The VFD indicates an active error
	        OR #sUDT_HMIStatus.CommunicationErrorMovikit;                          // The block generated an communication error

	    END_REGION

	    REGION 5.4 - Configuration Warning
	        //  Check if no faulty setup is active
	        //  This is the responcebility of the commisioning engineer

	        IF #iUDT_VfdConfig.PositionMax > #iUDT_VfdConfig.PositionMin          // Max position is bigger than min position
	            AND #iUDT_VfdConfig.PositionMax > 0                                // and not 0
	            AND #iUDT_VfdConfig.VFDSpeed > 0                                   // Max speed is not 0
	            AND #iUDT_VfdConfig.VFDAccDecel > 0                                // Maximum acceleration an deceleration time is not 0
	            AND "DB_ProfinetDiagnostic".ProfinetNetworks[#sUDT_PNDevice.PNNetworknumber].DeviceStatus[#sUDT_PNDevice.PNDeviceNumber].DeviceState.Configure
	        THEN
	            #sx_ConfigurationError := FALSE;                                    // Reset the configuration warning
	        ELSE
	            #sx_ConfigurationError := TRUE;                                     // Set configuration warning
	        END_IF;
	    END_REGION

	    REGION 5.5 - Common warning
	        // Set VFD warning active
	        #sx_WarningActive := #iUDT_VfdInputs.Status_Word_1.Warning             // The VFD indicates an active warning
	        OR #sUDT_HMIStatus.PositioningTimeOutError;                                 // The VFD did not reach the position in time.

	    END_REGION

	END_REGION

	REGION 6 - Check conditions to set VFD Ready signals

	    REGION 6.1 - Internal VFD ready

	        #sx_VFDReady := #sx_HardwareAvailable                                   // The hardware is powered up and detected
	        AND (#iUDT_VfdInputs.Status_Word_1.InverterReady                       // And VFD is ready to start
	        OR #sx_MotorRunning)                                                    // Or motor running
	        AND NOT #sx_ErrorActive                                                 // And no VFD error active
	        AND NOT #sx_ConfigurationError;
	        // AND NOT (#iqUDT_VSUInterface.PositionActual = #iqUDT_VSUInterface.RequestedPosition);    /// Commented out because  it was causing issues for the refernce drive                                // And no configuration error

	    END_REGION

	    REGION 6.2 - External VFD ready (to control)

	        #iqUDT_VSUInterface.Ready :=                                           // Signal ready is active if:
	        (#iqUDT_VSUInterface.Automatic                                         // And automatic mode request
	        AND NOT #iqUDT_VSUInterface.Manual                                     // And no manual mode request
	        AND #iUDT_VfdInputs.Status_Word_1.Referenced                           // And the drive is referenced
	        AND #iUDT_VfdInputs.Mode = 400)                                        // Actual application mode is equal to 400
	        OR
	        (NOT #iqUDT_VSUInterface.Automatic                                     // No automatic mode request
	        AND #iqUDT_VSUInterface.Manual                                         // AND manual mode request
	        AND #iUDT_VfdInputs.Mode = 100)                                        // And the actual application mode is equal to 100
	        OR
	        (#iqUDT_VSUInterface.Reference_command                                 // And the "refference" command is active
	        AND #iUDT_VfdInputs.Mode = 301)                                        // The actual application mode is equal TO 301
	        AND
	        (#sx_VFDReady                                                           // Status ready is active
	        AND #iqUDT_VSUInterface.RunEnabled);                                   // And running of the lifting device is enabled by VSU

	    END_REGION
	END_REGION

	REGION 7 - Set VFD control data

	    REGION 7.1 - Stop VFD

	        IF NOT #iqUDT_VSUInterface.Ready                                       // If VFD isn't ready to operate
	        THEN

	            #sx_StartVFD := FALSE;                                              // Reset start VFD
	            #qUDT_VfdOutputs.SetpointMode := 0;                                // Set the application mode to 0

	        END_IF;

	    END_REGION

	    REGION 7.3 - Reference VFD

	        IF #sx_VFDReady                                                         // If status VFD ready to operate is active
	            AND #iqUDT_VSUInterface.Reference_command                          // And the "refference" command is active
	        THEN

	            #qUDT_VfdOutputs.SetpointMode := 301;                              // Selecting FCB for reference travel FCB = 12

	            #tdi_EncoderPositionSetpoint := #iUDT_VfdConfig.Position[0];                                  // Set the position value as refference
	            #qUDT_VfdOutputs.SetpointPosition_hW := DINT_TO_WORD(SHR(IN := (#tdi_EncoderPositionSetpoint), N := 16));  // Send new position to encoder - high word
	            #qUDT_VfdOutputs.SetpointPosition_lW := DINT_TO_WORD(IN := #tdi_EncoderPositionSetpoint);                  // Send new position TO encoder - low word
	        END_IF;


	        IF #iqUDT_VSUInterface.Ready AND                                       // If VFD system is ready to operation
	            #iUDT_VfdInputs.Mode = 301                                         // And actual application mode  is equal to 301
	        THEN

	            #sx_StartVFD := TRUE;                                               // Set start VFD

	        END_IF;

	    END_REGION

	    REGION 7.4 - Manual mode - jogging

	        IF #sx_VFDReady                                                         // If status VFD ready to operation is active
	            AND #iqUDT_VSUInterface.Manual                                     // And manual mode request is active
	            AND NOT #iqUDT_VSUInterface.Automatic                              // And automatic mode request isn't active
	            AND #iqUDT_VSUInterface.RunEnabled                                 // And running of the lifting device is enabled by VSU
	            AND NOT #iqUDT_VSUInterface.Reference_command                      // And the "refference" command isn't active

	        THEN

	            #qUDT_VfdOutputs.SetpointMode := 100;                              // Selecting FCB for position-controlled jogging FCB = 20

	        END_IF;

	        // On position while jogging: stop, when button is released and pressed again continue to travel
	        //
	        #sR_TRIG_ManInPos(CLK := #sx_ManualPositionStop);

	        #sx_ManualPosHold := (#sx_ManualPosHold                                 // Hold movement as long as buttons are pressed
	        OR #sR_TRIG_ManInPos.Q)                                                // trigger position reached
	        AND (#iqUDT_VSUInterface.JogUp                                         // jogging up active
	        OR #iqUDT_VSUInterface.JogDown)                                        // jogging down active
	        AND #iqUDT_VSUInterface.Ready;                                         // ready to operate

	        // Jog commands

	        IF #iqUDT_VSUInterface.Ready                                           // If the VFD system is ready to operate
	            AND (#iUDT_VfdInputs.Mode = 100)                                   // And the actual application mode is equal to 100
	            AND #iqUDT_VSUInterface.JogUp                                      // And selected jog in positive direction
	            AND NOT #iqUDT_VSUInterface.JogDown                                // And not selected jog in negative direction
	            AND NOT #sx_ManualPosHold
	        THEN

	            #qUDT_VfdOutputs.Control_Word_1.JogPos := TRUE;                                                // Set jog positive VFD control bit
	            #qUDT_VfdOutputs.Control_Word_1.JogNeg := FALSE;                                               // Reset jog negative VFD control bit

	        ELSIF
	            #iqUDT_VSUInterface.Ready                                          // If the VFD system is ready to operate
	            AND (#iUDT_VfdInputs.Mode = 100)                                   // And the actual application mode is equal to 100
	            AND NOT #iqUDT_VSUInterface.JogUp                                  // And not selected jog in positive direction
	            AND #iqUDT_VSUInterface.JogDown                                    // And selected jog in negative direction
	            AND NOT #sx_ManualPosHold
	        THEN

	            #qUDT_VfdOutputs.Control_Word_1.JogPos := FALSE;                   // Reset jog positive VFD control bit
	            #qUDT_VfdOutputs.Control_Word_1.JogNeg := TRUE;                    // Set jog negative VFD control bit

	        ELSE

	            #qUDT_VfdOutputs.Control_Word_1.JogPos := FALSE;                   // Reset jog positive VFD control bit
	            #qUDT_VfdOutputs.Control_Word_1.JogNeg := FALSE;                   // Reset jog negative VFD control bit

	        END_IF;

	    END_REGION

	    REGION 7.5 - Automatic mode - for positioning

	        IF #sx_VFDReady                                                         // If status VFD ready to operation is active
	            AND #iqUDT_VSUInterface.Automatic                                  // And automatic mode request is active
	            AND NOT #iqUDT_VSUInterface.Manual                                 // And manual mode request isn't active
	            AND #iqUDT_VSUInterface.RunEnabled                                 // And running of the lifting device is enabled by VSU
	            AND #iUDT_VfdInputs.Status_Word_1.Referenced                       // And the drive is referenced
	            AND NOT #iqUDT_VSUInterface.Reference_command                      // And the "refference" command isn't active

	        THEN

	            #qUDT_VfdOutputs.SetpointMode := 400;                              // Select FCB for absolute positioning control FCB = 09

	        END_IF;

	        IF #iqUDT_VSUInterface.Ready AND                                       // IF VFD system is ready TO operation
	            #iUDT_VfdInputs.Mode = 400                                         // And actual application mode is equal to 400
	        THEN

	            #tdi_EncoderPositionSetpoint := #iUDT_VfdConfig.Position[#iqUDT_VSUInterface.PositionSetpoint];    // Move position request to setpoint postion
	            #qUDT_VfdOutputs.SetpointPosition_hW := DINT_TO_WORD(SHR(IN := (#tdi_EncoderPositionSetpoint), N := 16));         // Send new position to encoder - high word
	            #qUDT_VfdOutputs.SetpointPosition_lW := DINT_TO_WORD(IN := #tdi_EncoderPositionSetpoint);                         // Send new position to encoder - low word
	            #sx_StartVFD := TRUE;

	        END_IF;

	    END_REGION


	    REGION 7.6 - Set output speed

	        // When the drive was manual operated, first start in manual speed to go to position

	        #si_ManualSpeed := #ci_SpeedManualMode;                                 // Manual speed setpoint

	        IF (#iqUDT_VSUInterface.Manual                                          // Manual command is activated
	            OR #iqUDT_VSUInterface.GoReference)
	            AND NOT #iqUDT_VSUInterface.Automatic
	        THEN
	            #sx_RestartMan := TRUE;                                             // Set memory Manual was activated
	        END_IF;

	        IF #iqUDT_VSUInterface.PositionActual = #iqUDT_VSUInterface.PositionSetpoint     // Signal from VFD, indicating being in position
	            OR #iqUDT_VSUInterface.Automatic
	        THEN
	            #sx_RestartMan := FALSE;                                            // Reset memory Manual was activated
	        END_IF;


	        IF #iUDT_VfdInputs.Mode = 400                                          // If actual application mode is Auto ( 400 )
	        THEN
	            IF NOT #sx_RestartMan                                               // Manual was not activated

	            THEN
	                #qUDT_VfdOutputs.SetpointSpeed := #iUDT_VfdConfig.VFDSpeed;   // Move speedsetpoint to output
	            ELSE                                                                // If manual was activated then
	                #qUDT_VfdOutputs.SetpointSpeed := #si_ManualSpeed;             // Move manual speedsetpoint to output
	            END_IF;

	        ELSIF #iUDT_VfdInputs.Mode = 100                                       // If actual application mode is manual ( 100 )
	        THEN

	            #qUDT_VfdOutputs.SetpointSpeed := #si_ManualSpeed;                 // Move manual speedsetpoint TO output

	        END_IF;

	    END_REGION


	    REGION 7.8 - Other control signals to VFD

	        #qUDT_VfdOutputs.Control_Word_1.EnableRapidStop := (#sx_HardwareAvailable AND #iqUDT_VSUInterface.RunEnabled); // Writing states of VFD power is ready or simulation to enable VFD to run
	        #qUDT_VfdOutputs.Control_Word_1.EnableApplicationStop := #sx_VFDReady AND ((NOT (#sdi_ActualPositionValue = #tdi_EncoderPositionSetpoint) AND #iqUDT_VSUInterface.Automatic) OR (#iqUDT_VSUInterface.Manual AND ((#iqUDT_VSUInterface.JogDown OR #iqUDT_VSUInterface.JogUp) OR #iqUDT_VSUInterface.Reference_command)));                             // Writing state to enable VFD operation
	        #qUDT_VfdOutputs.Control_Word_1.ReleaseBrake := FALSE;                                             // Not used
	        #qUDT_VfdOutputs.Control_Word_1.ApplyRelativePositioning := FALSE;                                 // Not used for speed control
	        #qUDT_VfdOutputs.Control_Word_1.StartStop := #sx_StartVFD;                                         // Writing state to start or stop VFD
	        #qUDT_VfdOutputs.Control_Word_1.ResetError := #iqUDT_VSUInterface.InternalErrorReset;             // Reseting VFD errors with error reset bit
	        #qUDT_VfdOutputs.Control_Word_1.ActivateDriveTrain2 := FALSE;                                      // Not used for MoviGear with on Drive Train
	        #qUDT_VfdOutputs.Control_Word_1.DeactivateSW_LimitSwitch := FALSE;                                 // Not used
	        #qUDT_VfdOutputs.Control_Word_1.ActivateInhibit := NOT #sx_VFDReady;                                // Controller Inhibit has to be "false" before start/stop
	        #qUDT_VfdOutputs.Control_Word_1.ActivateStandby := FALSE;                                          // Not used
	        #qUDT_VfdOutputs.Control_Word_1.MovikitHandshakeIn := #sx_MovikitHandshakeIn;                      // Set "MoviKit" handshake input to 1 by 0.5 sec.

	    END_REGION

	    REGION 7.9 - Acceleration and deceleration ramps

	        #qUDT_VfdOutputs.SetpointAcceleration := #iUDT_VfdConfig.VFDAccDecel;
	        #qUDT_VfdOutputs.SetpointDeceleration := #iUDT_VfdConfig.VFDAccDecel;

	    END_REGION

	END_REGION

	REGION 8 - In case of communication error reset VFD outputs

	    IF NOT #sx_HardwareAvailable                                                                            // If hardware is not available

	    THEN

	        #qUDT_VfdOutputs.Control_Word_1.ResetError := FALSE;                                               // Reset reset VFD error
	        #qUDT_VfdOutputs.Control_Word_1.ActivateDriveTrain2 := FALSE;                                      // Reset activate drive train
	        #qUDT_VfdOutputs.Control_Word_1.DeactivateSW_LimitSwitch := FALSE;                                 // Reset deactivate software limit switch
	        #qUDT_VfdOutputs.Control_Word_1.ActivateInhibit := FALSE;                                          // Reset activate inhibit
	        #qUDT_VfdOutputs.Control_Word_1.ActivateStandby := FALSE;                                          // Reset activate standby
	        #qUDT_VfdOutputs.Control_Word_1.MovikitHandshakeIn := FALSE;                                       // Reset movikit hanshake input
	        #qUDT_VfdOutputs.Control_Word_1.EnableRapidStop := FALSE;                                          // Reset enable rapid stop
	        #qUDT_VfdOutputs.Control_Word_1.EnableApplicationStop := FALSE;                                    // Reset enable application stop
	        #qUDT_VfdOutputs.Control_Word_1.ReleaseBrake := FALSE;                                             // Reset release brake
	        #qUDT_VfdOutputs.Control_Word_1.JogPos := FALSE;                                                   // Reset jog in positive direction
	        #qUDT_VfdOutputs.Control_Word_1.JogNeg := FALSE;                                                   // Reset jog in negative direction
	        #qUDT_VfdOutputs.Control_Word_1.ApplyRelativePositioning := FALSE;                                 // Reset applying relatice positioning
	        #qUDT_VfdOutputs.Control_Word_1.StartStop := FALSE;                                                // Reset Start/Stop VFD
	    END_IF;
	END_REGION

	REGION 9 - Statistics

	    // Number OF times the VFD had an internal error

	    #sR_TRIG_PNSlaveNotOnline(CLK := #sUDT_HMIStatus.PNSlaveNotOnline);       // Detect the rising edge of the error

	    IF #iqUDT_VSUInterface.ResetStatistics OR                                  // If there is signal to reset statistics from VSU interface
	        #sUDT_HMIStatus.PNSlaveNotOnline                                       // Or the error occured
	    THEN

	        "FC_Statistics"(ix_Reset := #iqUDT_VSUInterface.ResetStatistics,       // Reset statistics
	                        ix_Activate := #sUDT_HMIStatus.PNSlaveNotOnline,       // Actual error
	                        ix_RTrigActivate := #sR_TRIG_PNSlaveNotOnline.Q,       // Trigger rising edge error
	                        iqUDT_Statistics := #iqUDT_VFDStatistics.PNSlaveNotOnline);   // Statistics structure
	    END_IF;

	    // Number of ethernet communication faults to VFD drive

	    #sR_TRIG_PNSlaveError(CLK := #sUDT_HMIStatus.PNSlaveError);               // Detect the rising edge of the error
	    IF #iqUDT_VSUInterface.ResetStatistics OR                                  // If there is signal to reset statistics from VSU interface
	        #sUDT_HMIStatus.PNSlaveError                                           // Or the error occured
	    THEN

	        "FC_Statistics"(ix_Reset := #iqUDT_VSUInterface.ResetStatistics,       // Reset statistics
	                        ix_Activate := #sUDT_HMIStatus.PNSlaveError,           // Actual error
	                        ix_RTrigActivate := #sR_TRIG_PNSlaveError.Q,           // Trigger rising edge error
	                        iqUDT_Statistics := #iqUDT_VFDStatistics.PNSlaveError);       // Statistics structure

	    END_IF;


	    // Number of times the VFD had an internal error

	    #sR_TRIG_InternalError(CLK := #sUDT_HMIStatus.InternalError);             // Detect the rising edge of the error

	    IF #iqUDT_VSUInterface.ResetStatistics OR                                  // IF there is signal TO reset statistics from VSU interface
	        #sUDT_HMIStatus.InternalError                                          // Or the error occured
	    THEN

	        "FC_Statistics"(ix_Reset := #iqUDT_VSUInterface.ResetStatistics,       // Reset statistics
	                        ix_Activate := #sUDT_HMIStatus.InternalError,          // Actual error
	                        ix_RTrigActivate := #sR_TRIG_InternalError.Q,          // Trigger rising edge error
	                        iqUDT_Statistics := #iqUDT_VFDStatistics.VFDInternalError);       // Statistics structure

	    END_IF;

	    // Number OF times the VFD had a safety error

	    #sR_TRIG_CommunicationErrorMovikit(CLK := #sUDT_HMIStatus.CommunicationErrorMovikit); // Detect the rising edge of the error

	    IF #iqUDT_VSUInterface.ResetStatistics OR                                  // If there is signal to reset statistics from VSU interface
	        #sUDT_HMIStatus.CommunicationErrorMovikit                              // Or the error occured
	    THEN

	        "FC_Statistics"(ix_Reset := #iqUDT_VSUInterface.ResetStatistics,       // Reset statistics
	                        ix_Activate := #sUDT_HMIStatus.CommunicationErrorMovikit,              // Actual error
	                        ix_RTrigActivate := #sR_TRIG_CommunicationErrorMovikit.Q,              // Trigger rising edge error
	                        iqUDT_Statistics := #iqUDT_VFDStatistics.CommunicationErrorMovikit);  // Statistics structure

	    END_IF;

	    // Number of times the VFD has been running

	    #sR_TRIG_Running(CLK := #iUDT_VfdInputs.Status_Word_1.DriveActive);       // Detect the rising edge of the signal

	    IF #iqUDT_VSUInterface.ResetStatistics OR                                  // If there is signal to reset statistics from VSU interface
	        #iUDT_VfdInputs.Status_Word_1.STO_Inactive                             // Or the status occured
	    THEN

	        "FC_Statistics"(ix_Reset := #iqUDT_VSUInterface.ResetStatistics,       // Reset statistics
	                        ix_Activate := #iUDT_VfdInputs.Status_Word_1.DriveActive,  // Actual status
	                        ix_RTrigActivate := #sR_TRIG_Running.Q,                // Trigger rising edge
	                        iqUDT_Statistics := #iqUDT_VFDStatistics.Running);    // Statistics structure

	    END_IF;
	END_REGION

	REGION 10 - Write interface outputs

	    //Internal Error
	    #iqUDT_VSUInterface.InternalErrorVFD := #sx_ErrorActive;                   // Set the internal VFD error bit in VSU interface IF Any fault is active

	    //Internal Warning
	    #iqUDT_VSUInterface.InternalWarningVFD := #sx_WarningActive;               // Set the internal VFD warning bit if any warning is active

	    //Motor running
	    #iqUDT_VSUInterface.MotorRunning := #iUDT_VfdInputs.Status_Word_1.DriveActive;    // Set motor is running in VSU interface IF status control Word "motor running" is active

	    //Send signal VFD is referenced
	    #iqUDT_VSUInterface.Referenced := #iUDT_VfdInputs.Status_Word_1.Referenced;       // Write state of drive is referenced from VFD to VSU interface


	    #iqUDT_VSUInterface.Positioning := #iqUDT_VSUInterface.PositionSetpoint <> #iqUDT_VSUInterface.PositionActual  // Set the lifting device is positioning if position setpoint is different than actual position
	    AND #iqUDT_VSUInterface.Automatic                                      // AND automatic mode enabled
	    AND NOT #iqUDT_VSUInterface.InternalErrorVFD;                          // And internal error VFD no occurred

	    #iqUDT_VSUInterface.StartLowSpeed := #sx_RestartMan;                       // Indicating to VSU the VSD is starting in low speed

	    #qUDT_HMIStatus := #sUDT_HMIStatus;                                       // Copy status to output
	END_REGION

	REGION 11 - error codes
	    (*
	    FCB number |                       | Meaning
	    ______________________________________________________________________________________________________________
	        1                               Output stage inhibit
	        2                               Default stop
	        4                               Manual Mode
	        5                               Speed control
	                101                     Speed-controlled jogging. Encoder feedback NOT required.
	                200                     Speed control. Encoder feedback NOT required.
	        6                               Interpolated speed control
	        7                               Torque control
	        8                               Interpolated torque control
	        9                               Positioning mode
	                400                     Absolute position control
	                401                     Relative position control
	                402                     Modulo position control - positive
	                403                     Modulo position control - negative
	                404                     Modulo position control - shortest distance
	        10                              Interpolated position control
	        12                              Referencing mode
	                300                     Reference travel - offset via parameter
	                301                     Reference travel - offset via fieldbus
	        13                              Stop at application limits
	        14                              Emergency stop
	        18                              Rotor position identification
	        19                              Position hold control
	        20                              Jog mode
	                100                     Position-controlled jogging. Encoder feedback required
	        21                              Brake test
	        25                              Motor parameter measurement
	        26                              Stop at user limits


	    Error code | Suberror code        | Meaning                                | Measure
	    ______________________________________________________________________________________________________________
	        3       1                       Ground fault                            Consult "Fault table" in
	        4       1                       Brake chopper fault                     document 'SEW Movigear-C 25887130.PDF'
	        6       1                       Line fault                              Chapter 8.7
	        7       1                       DC link fault
	        8       1,2,3                   Speed monitoring fault
	        9       1,2,5,6,9,10            Control mode fault
	        10      1,3-11                  Data flexibility fault
	        11      1-6                     Temperature monitoring fault
	        12      1,2                     Fault brake
	        13      5,24                    Encoder 1 fault
	        16      5-8,10,20-27            Startup fault
	        19      1-9                     Process data fault
	        20      2,11                    Fault device monitoring
	        23      4                       Power section fault
	        25      2-7,20,21,30,31,61,70   Parameter memory monitoring
	        26      1,3                     External fault
	        28      1-12,14                 FCB drive function fault
	        29      1-4                     Hardware limit switch fault
	        30      1-3                     Software limit switch fault
	        31      1-4,7,9                 Thermal protection fault
	        32      2-6,12                  Communication fault
	        33      11,12,13                system initialisation fault
	        34      1                       Process data configuration fault
	        35      1-5                     Function activation fault
	        42      1-3                     Lag fault
	        46      2,3,50,51,52            Safety card fault
	        51      1                       Analog processing fault

	    Error code | Suberror code        | Meaning                                | Measure
	    ______________________________________________________________________________________________________________
	        1       1,2                     Output stage monitoring fault           Contact SEW-Eurodrive Service
	        4       2                       Brake chopper fault
	        7       2                       DC link fault
	        9       3,4,8                   Control mode fault
	        10      2,99                    Data flexibility fault
	        11      7,8                     Temperature monitoring fault
	        13      1,3,6,7.8,9,11,13,      Encoder 1 fault
	                15,22,23
	        16      2,11,12,30              Startup fault
	        17      7                       Internal processor fault
	        18      1,3,4,7,8,9,10,12,13    Software fault
	        20      1,7                     Fault device monitoring
	        21      1                       S-Drive 1 fault
	        23      5,6,7,8                 Power section fault
	        25      10,12-19,50,51,81       Parameter memory monitoring
	        28      13                      FCB drive funcyio fault
	        33      1,2,6,7,8,10            System initialisation fault
	        46      1                       Safety card fault

	    Function Control Block (FCB) codes
	    FBC = 01 Output stage inhibit
	    FBC = 02 Default stop
	    FBC = 04 Manual Mode
	    FBC = 05 Speed control
	     101 - Speed-controlled jogging. Encoder feedback NOT required.
	     200 - Speed control. Encoder feedback NOT required.
	    FBC = 06 Interpolated speed control
	    FBC = 07 Torque control
	    FBC = 08 Interpolated torque control
	    FBC = 09 Positioning mode
	    400 - Absolute position control
	    401 - Relative position control
	    402 - Modulo position control - positive
	    403 - Modulo position control - negative
	    404 - Modulo position control - shortest distance
	    FBC = 10 Interpolated position control
	    FBC = 12 Referencing mode
	    300 - Reference travel - offset via parameter
	    301 - Reference travel - offset via fieldbus
	    FBC = 13 Stop at application limits
	    FBC = 14 Emergency stop
	    FBC = 18 Rotor position identification
	    FBC = 19 Position hold control
	    FBC = 20 Jog mode
	     100 - Position-controlled jogging. Encoder feedback required
	    FBC = 21 Brake test
	    FBC = 25 Motor parameter measurement
	    FBC = 26 Stop at user limits

	    *)
	END_REGION
END_FUNCTION_BLOCK

FUNCTION_BLOCK "FB_RIOVSU"
TITLE = FB_RIOVSU
{ S7_Optimized_Access := 'TRUE' }
AUTHOR : MHSE
FAMILY : GeneralSystemFunctions
VERSION : 3.0
// ATTRIBUTES
// AUTO_NUMBER = True
// BLOCK_NUMBER = 226
// END_ATTRIBUTES
   VAR_INPUT
      is_ET200spPNDeviceName { ExternalAccessible := 'False'; ExternalVisible := 'False'; ExternalWritable := 'False'} : String;   //   Name of the ET200sp device
      ix_400VintOk { ExternalAccessible := 'False'; ExternalVisible := 'False'; ExternalWritable := 'False'} : Bool;   //   TRUE if internal circuit breaker 400V is ok
      ix_400VextOk { ExternalAccessible := 'False'; ExternalVisible := 'False'; ExternalWritable := 'False'} : Bool;   //   TRUE if external 400V Main cabinet is ok
      ix_BrakeSupplyOk { ExternalAccessible := 'False'; ExternalVisible := 'False'; ExternalWritable := 'False'} : Bool;   //   TRUE if circuit breaker of brake power supply is ok
      ix_ThermalBrake { ExternalAccessible := 'False'; ExternalVisible := 'False'; ExternalWritable := 'False'} : Bool;   //   TRUE when No thermal error
      ix_24VOk { ExternalAccessible := 'False'; ExternalVisible := 'False'; ExternalWritable := 'False'} : Bool;   //   TRUE when 24V power supply to RIO is ok
      ix_SimulationModeActive { ExternalAccessible := 'False'; ExternalVisible := 'False'; ExternalWritable := 'False'} : Bool;   //   True when Simulation mode active
      ix_HardwareOk { ExternalAccessible := 'False'; ExternalVisible := 'False'; ExternalWritable := 'False'} : Bool;   //  TRUE when  hardware is Ok
   END_VAR

   VAR_OUTPUT
      qUDT_HMIStatus { ExternalAccessible := 'False'; ExternalVisible := 'False'; ExternalWritable := 'False'} : "UDT_RIOVSUStatus";   //   HMI status structure
   END_VAR

   VAR_IN_OUT
      iqUDT_Statistics : "UDT_RIOVSUStatistics";   //   Statistics structure
      iqUDT_VSUInterface : "UDT_VSUInterface";   //   Interface RIO and VSU
   END_VAR

   VAR
      sUDT_HMIStatus { ExternalAccessible := 'False'; ExternalVisible := 'False'; ExternalWritable := 'False'; S7_SetPoint := 'False'} : "UDT_RIOVSUStatus";   //   HMI status structure
      sUDT_PNDevice { ExternalAccessible := 'False'; ExternalVisible := 'False'; ExternalWritable := 'False'; S7_SetPoint := 'False'} : "UDT_PNDevice";   //   PN device structure
      sa_PNPortsStatus { ExternalAccessible := 'False'; ExternalVisible := 'False'; ExternalWritable := 'False'} : Array[1..8] of Bool;   // TRUE when specific port has an error
      sFB_TimerOnOffDelayCheckSupply { ExternalAccessible := 'False'; ExternalVisible := 'False'; ExternalWritable := 'False'; S7_SetPoint := 'False'} : "FB_TimerOnOffDelay";   //   MHS "TimerOnOffDelay" - to delay time for VFD supply contactor
      sR_TRIG_Int400VCBError {InstructionName := 'R_TRIG'; LibVersion := '1.0'; ExternalAccessible := 'False'; ExternalVisible := 'False'; ExternalWritable := 'False'; S7_SetPoint := 'False'} : R_TRIG;   //   Rising edge for trigger 400v internal error
      sR_TRIG_Int24VError {InstructionName := 'R_TRIG'; LibVersion := '1.0'; ExternalAccessible := 'False'; ExternalVisible := 'False'; ExternalWritable := 'False'; S7_SetPoint := 'False'} : R_TRIG;   //   Rising edge for trigger 24v internal error
      sR_TRIG_BrakeCBerror {InstructionName := 'R_TRIG'; LibVersion := '1.0'; ExternalAccessible := 'False'; ExternalVisible := 'False'; ExternalWritable := 'False'; S7_SetPoint := 'False'} : R_TRIG;   //   Rising edge for trigger brake circuit breaker tripped
      sR_TRIG_BrakeThermError {InstructionName := 'R_TRIG'; LibVersion := '1.0'; ExternalAccessible := 'False'; ExternalVisible := 'False'; ExternalWritable := 'False'; S7_SetPoint := 'False'} : R_TRIG;   //   Rising edge for trigger brake thermal error
      sR_TRIG_DeviceFound {InstructionName := 'R_TRIG'; LibVersion := '1.0'; ExternalAccessible := 'False'; ExternalVisible := 'False'; ExternalWritable := 'False'; S7_SetPoint := 'False'} : R_TRIG;   //   Rising edge for trigger scan modules
      sR_TRIG_PNSlaveNotOnline {InstructionName := 'R_TRIG'; LibVersion := '1.0'; ExternalAccessible := 'False'; ExternalVisible := 'False'; ExternalWritable := 'False'; S7_SetPoint := 'False'} : R_TRIG;   //   Rising edge for trigger Profinet slave not online statistics
      sR_TRIG_PNSlaveError {InstructionName := 'R_TRIG'; LibVersion := '1.0'; ExternalAccessible := 'False'; ExternalVisible := 'False'; ExternalWritable := 'False'; S7_SetPoint := 'False'} : R_TRIG;   //   Rising edge for trigger Profinet slave error statistics
      si_ModuleStateReturn { ExternalAccessible := 'False'; ExternalVisible := 'False'; ExternalWritable := 'False'} : Int;   //   Status structure
      si_NrOfModulesWithError { ExternalAccessible := 'False'; ExternalVisible := 'False'; ExternalWritable := 'False'} : Int;   //   Number of the faulty modules
      sx_PNSlaveOnline { ExternalAccessible := 'False'; ExternalVisible := 'False'; ExternalWritable := 'False'} : Bool;   //   Profinet device is online and error free
      sx_PowerOk { ExternalAccessible := 'False'; ExternalVisible := 'False'; ExternalWritable := 'False'} : Bool;   //   True = External Power OK
      sx_ConfigurationError { ExternalAccessible := 'False'; ExternalVisible := 'False'; ExternalWritable := 'False'} : Bool;   //   Commissioning: configuration error
   END_VAR

   VAR_TEMP
      ta_Configured : Array[0..127] of Bool;   //   Configured modules array
      ta_Exist : Array[0..127] of Bool;   //   Existing modules array
      ta_Error : Array[0..127] of Bool;   //   Faulty modules array
      ti_NrOfModule : Int;   //   Number of current module
      ti_DiagArraySize : Int;   //   Diagnostic array size
   END_VAR

   VAR CONSTANT
      cui_ConfiguredModulesMode : UInt := 1;   //   Mode selector: 1 = Configured modules scan mode
      cui_ModuleErrorMode : UInt := 2;   //   Mode selector: 2 = Existing modules scan mode
      cui_ExistingModulesMode : UInt := 4;   //   Mode selector: 3 = Module Error scan mode
      ci_PowerSupplyDelayTime : UInt := 4000;   //   Power supply delay time
      ci_NumberOfProfinetPorts : Int := 2;   // Number of Profinet ports in device
   END_VAR


BEGIN
	(*
	----------------------------------------------------------------------------------------

	Version history:
	Date        | Version   | Author        | Remark
	----------------------------------------------------------------------------------------
	03/09-2019  | 2.1       | F.Baten       | first release MHS TIA 15.1
	23/09/2019  | 2.2       | F.Baten       | Changed region 1 contents to FC
	12/10/2019  | 2.3       | L. Klar       | Updated status structure
	14/10/2019  | 2.4       | S. Deulkar    | Added equipment control structure and created
	                                        | region for status
	12/11/2019  | 3.0       | P.Majka       | 3.0 MHS library release TIA 15.1
	29/11/2019  | 3.1       | F.Baten       | Updated interface to VSU
	04/12/2019  | 3.2       | F.Baten       | Region 3: ix_SimulationModeActive rearranged to correct position
	09/12/2019  | 3.3       | F.Baten       | Region 5: added #ix_SimulationModeActive to PNDeviceOk
	04/03/2020  | 3.4       | F.Baten       | Updated errors and warnings and interface to VSU
	06/08/2020  | 3.5       | L.Klar        | Initialize the #si_NrOfModulesWithError on the reset
	03/11/2020  | 3.9       | K.Pokorski    | Profinet ports diagnostics added
	02/08/2021  | 3.5       | S. Deulkar    | Added logic to reset error when 24V is not okay.
	21/02/2023  | 4.0       | F.Baten       | 4.0 Release TIA 17.5
	*)

	REGION 1 - Get Device Profinet information

	    "FC_GetDevicePN"(is_PNDeviceName := #is_ET200spPNDeviceName,
	                     ix_SimulationModeActive := #ix_SimulationModeActive,
	                     iqUDT_PND := #sUDT_PNDevice);


	    "FC_GetPNPortStatus"(ii_NumberOfPorts := #ci_NumberOfProfinetPorts,
	                         iUDT_DevicePNInfo := #sUDT_PNDevice,
	                         qa_PortFault => #sa_PNPortsStatus);

	END_REGION

	REGION 2 - Reset errors
	    // reset Profinet Slave error/not online
	    IF #iqUDT_VSUInterface.InternalErrorReset
	        OR NOT #ix_24VOk
	    THEN
	        #sUDT_HMIStatus."400VCircuitBreaker" := FALSE;
	        #sUDT_HMIStatus.BrakeCircuitBreaker := FALSE;
	        #sUDT_HMIStatus.BrakeThermalError := FALSE;
	        #sUDT_HMIStatus.PNSlaveNotOnline := FALSE;
	        #sUDT_HMIStatus.PNSlaveError := FALSE;
	        #sUDT_HMIStatus."24VPowersupplyError" := FALSE;
	        #sUDT_HMIStatus.PNSlaveWarning := FALSE;
	        #si_NrOfModulesWithError := 0;

	    END_IF;

	    // reset ET200sp module error status
	    IF #sUDT_HMIStatus.PNSlaveNotOnline OR #iqUDT_VSUInterface.InternalErrorReset OR NOT #ix_24VOk
	    THEN
	        FILL_BLK(IN := FALSE,
	                 COUNT := 32,
	                 OUT => #sUDT_HMIStatus.ET200sp_ErrorModule[0]);
	    END_IF;

	END_REGION

	REGION 3 - Update PN slave device status
	    // Hardware will only be available after the delay, so the device has time for the initialisation
	    #sFB_TimerOnOffDelayCheckSupply(iudi_OnDelayTime := #ci_PowerSupplyDelayTime,
	                                    ix_SignalToDelay := #ix_24VOk,
	                                    qx_DelayedSignal => #sx_PowerOk);

	    // check if PN device is online
	    IF ((NOT "DB_ProfinetDiagnostic".ProfinetNetworks[#sUDT_PNDevice.PNNetworknumber].DeviceStatus[#sUDT_PNDevice.PNDeviceNumber].DeviceState.Exist
	        AND #sx_PowerOk)
	        OR NOT #sUDT_PNDevice.PNDeviceFound)
	        AND NOT #ix_SimulationModeActive
	    THEN
	        #sUDT_HMIStatus.PNSlaveNotOnline := TRUE;
	    END_IF;

	    // Check if PN ports are healthy
	    IF #sa_PNPortsStatus[1] XOR #sa_PNPortsStatus[2] THEN
	        #sUDT_HMIStatus.PNSlaveWarning := TRUE;
	    END_IF;

	    // check if PN device has an error
	    IF "DB_ProfinetDiagnostic".ProfinetNetworks[#sUDT_PNDevice.PNNetworknumber].DeviceStatus[#sUDT_PNDevice.PNDeviceNumber].DeviceState.Error
	        AND #sx_PowerOk
	        AND NOT #ix_SimulationModeActive
	        AND NOT #sUDT_HMIStatus.PNSlaveWarning

	    THEN
	        #sUDT_HMIStatus.PNSlaveError := TRUE;
	    END_IF;

	    // set bit when PN device is healthy (online and no error)
	    #sx_PNSlaveOnline := NOT #sUDT_HMIStatus.PNSlaveNotOnline
	    AND #sUDT_PNDevice.PNDeviceFound
	    AND #sx_PowerOk
	    OR #ix_SimulationModeActive;

	    // create rising edge to scan module status when device is found
	    #sR_TRIG_DeviceFound(CLK := #sUDT_PNDevice.PNDeviceFound);

	END_REGION

	REGION 4 - Status update modules ET200sp
	    // update ET200sp module status
	    IF (#sx_PNSlaveOnline
	        AND (#sUDT_HMIStatus.PNSlaveError
	        OR #sUDT_HMIStatus.PNSlaveWarning))
	        OR #sR_TRIG_DeviceFound.Q
	    THEN
	        // get configured modules
	        #si_ModuleStateReturn := ModuleStates(LADDR := "DB_ProfinetDiagnostic".ProfinetNetworks[#sUDT_PNDevice.PNNetworknumber].DeviceStatus[#sUDT_PNDevice.PNDeviceNumber].DeviceState.HW_ID,
	                                              MODE := #cui_ConfiguredModulesMode,
	                                              STATE := #ta_Configured);

	        // get module online status
	        #si_ModuleStateReturn := ModuleStates(LADDR := "DB_ProfinetDiagnostic".ProfinetNetworks[#sUDT_PNDevice.PNNetworknumber].DeviceStatus[#sUDT_PNDevice.PNDeviceNumber].DeviceState.HW_ID,
	                                              MODE := #cui_ExistingModulesMode,
	                                              STATE := #ta_Exist);

	        // get module error status
	        #si_ModuleStateReturn := ModuleStates(LADDR := "DB_ProfinetDiagnostic".ProfinetNetworks[#sUDT_PNDevice.PNNetworknumber].DeviceStatus[#sUDT_PNDevice.PNDeviceNumber].DeviceState.HW_ID,
	                                              MODE := #cui_ModuleErrorMode,
	                                              STATE := #ta_Error);

	        // Handle ET200sp module errors/offline
	        IF (#si_ModuleStateReturn = 0)
	        THEN
	            #si_NrOfModulesWithError := 0;

	            #ti_DiagArraySize := "FC_GetNrOfArrayEl"(iv_Array := "DB_ProfinetDiagnostic".ProfinetNetworks[#sUDT_PNDevice.PNNetworknumber].DeviceStatus[#sUDT_PNDevice.PNDeviceNumber].Module);

	            FOR #ti_NrOfModule := 0 TO (#ti_DiagArraySize - 1) DO

	                // check if the module is configured
	                IF (#ta_Configured[#ti_NrOfModule])
	                THEN
	                    "DB_ProfinetDiagnostic".ProfinetNetworks[#sUDT_PNDevice.PNNetworknumber].DeviceStatus[#sUDT_PNDevice.PNDeviceNumber].Module[#ti_NrOfModule].Configured := TRUE;
	                    // and check if the module is online
	                    IF (#ta_Exist[#ti_NrOfModule])
	                    THEN
	                        "DB_ProfinetDiagnostic".ProfinetNetworks[#sUDT_PNDevice.PNNetworknumber].DeviceStatus[#sUDT_PNDevice.PNDeviceNumber].Module[#ti_NrOfModule].Exist := TRUE;

	                    ELSE
	                        "DB_ProfinetDiagnostic".ProfinetNetworks[#sUDT_PNDevice.PNNetworknumber].DeviceStatus[#sUDT_PNDevice.PNDeviceNumber].Module[#ti_NrOfModule].Exist := FALSE;
	                        #sUDT_HMIStatus.ET200sp_ErrorModule[#ti_NrOfModule] := TRUE;
	                        // count number of modules with error/offline
	                        #si_NrOfModulesWithError += 1;
	                    END_IF;

	                    // and check if the module has an error
	                    IF (NOT #ta_Error[#ti_NrOfModule])
	                    THEN
	                        "DB_ProfinetDiagnostic".ProfinetNetworks[#sUDT_PNDevice.PNNetworknumber].DeviceStatus[#sUDT_PNDevice.PNDeviceNumber].Module[#ti_NrOfModule].Error := FALSE;

	                    ELSE
	                        "DB_ProfinetDiagnostic".ProfinetNetworks[#sUDT_PNDevice.PNNetworknumber].DeviceStatus[#sUDT_PNDevice.PNDeviceNumber].Module[#ti_NrOfModule].Error := TRUE;
	                        #sUDT_HMIStatus.ET200sp_ErrorModule[#ti_NrOfModule] := TRUE;
	                        // count number OF modules with error/offline
	                        #si_NrOfModulesWithError += 1;
	                    END_IF;

	                ELSE
	                    // reset module status when module is not configured
	                    "DB_ProfinetDiagnostic".ProfinetNetworks[#sUDT_PNDevice.PNNetworknumber].DeviceStatus[#sUDT_PNDevice.PNDeviceNumber].Module[#ti_NrOfModule].Configured := FALSE;
	                    "DB_ProfinetDiagnostic".ProfinetNetworks[#sUDT_PNDevice.PNNetworknumber].DeviceStatus[#sUDT_PNDevice.PNDeviceNumber].Module[#ti_NrOfModule].Exist := FALSE;
	                    "DB_ProfinetDiagnostic".ProfinetNetworks[#sUDT_PNDevice.PNNetworknumber].DeviceStatus[#sUDT_PNDevice.PNDeviceNumber].Module[#ti_NrOfModule].Error := FALSE;

	                END_IF;
	            END_FOR;
	        END_IF;
	    END_IF;

	END_REGION

	REGION 5 - Check RIO Panel Status

	    // create 400v internal error
	    IF NOT #ix_400VintOk
	    THEN
	        #sUDT_HMIStatus."400VCircuitBreaker" := TRUE;
	    END_IF;

	    // create error circuit breaker brake tripped
	    IF NOT #ix_BrakeSupplyOk
	    THEN
	        #sUDT_HMIStatus.BrakeCircuitBreaker := TRUE;
	    END_IF;

	    // Create error thermal overload brake
	    IF NOT #ix_ThermalBrake
	    THEN
	        #sUDT_HMIStatus.BrakeThermalError := TRUE;
	    END_IF;

	    // Create error thermal overload brake
	    IF NOT #ix_24VOk
	    THEN
	        #sUDT_HMIStatus."24VPowersupplyError" := TRUE;
	    END_IF;

	    // check if 400 v to VFD positioning is ok
	    #iqUDT_VSUInterface.VSUMainPowerOk := #ix_400VextOk;

	    // set config not ok bit if no device found
	    #sx_ConfigurationError := NOT #sUDT_PNDevice.PNDeviceFound;

	END_REGION

	REGION 6 - Statistics
	    // create trigger on error and create statistics
	    #sR_TRIG_Int400VCBError(CLK := #sUDT_HMIStatus."400VCircuitBreaker");

	    IF #iqUDT_VSUInterface.ResetStatistics OR #sUDT_HMIStatus."400VCircuitBreaker"
	    THEN

	        "FC_Statistics"(ix_Reset := #iqUDT_VSUInterface.ResetStatistics,
	                        ix_Activate := #sUDT_HMIStatus."400VCircuitBreaker",
	                        ix_RTrigActivate := #sR_TRIG_Int400VCBError.Q,
	                        iqUDT_Statistics := #iqUDT_Statistics.Int400VCBError);
	    END_IF;

	    // create trigger on error and create statistics
	    #sR_TRIG_Int24VError(CLK := #sUDT_HMIStatus."24VPowersupplyError");

	    IF #iqUDT_VSUInterface.ResetStatistics OR #sUDT_HMIStatus."24VPowersupplyError"
	    THEN

	        "FC_Statistics"(ix_Reset := #iqUDT_VSUInterface.ResetStatistics,
	                        ix_Activate := #sUDT_HMIStatus."24VPowersupplyError",
	                        ix_RTrigActivate := #sR_TRIG_Int24VError.Q,
	                        iqUDT_Statistics := #iqUDT_Statistics."24VError");
	    END_IF;

	    // create trigger on error and create statistics
	    #sR_TRIG_BrakeCBerror(CLK := #sUDT_HMIStatus.BrakeCircuitBreaker);

	    IF #iqUDT_VSUInterface.ResetStatistics OR #sUDT_HMIStatus.BrakeCircuitBreaker
	    THEN

	        "FC_Statistics"(ix_Reset := #iqUDT_VSUInterface.ResetStatistics,
	                        ix_Activate := #sUDT_HMIStatus.BrakeCircuitBreaker,
	                        ix_RTrigActivate := #sR_TRIG_BrakeCBerror.Q,
	                        iqUDT_Statistics := #iqUDT_Statistics.BrakeCBerror);
	    END_IF;

	    // create trigger on error and create statistics
	    #sR_TRIG_BrakeThermError(CLK := #sUDT_HMIStatus.BrakeThermalError);

	    IF #iqUDT_VSUInterface.ResetStatistics OR #sUDT_HMIStatus.BrakeThermalError
	    THEN

	        "FC_Statistics"(ix_Reset := #iqUDT_VSUInterface.ResetStatistics,
	                        ix_Activate := #sUDT_HMIStatus.BrakeThermalError,
	                        ix_RTrigActivate := #sR_TRIG_BrakeThermError.Q,
	                        iqUDT_Statistics := #iqUDT_Statistics.BrakeThermError);
	    END_IF;

	    // create trigger on error and create statistics for profinet slave not online
	    #sR_TRIG_PNSlaveNotOnline(CLK := #sUDT_HMIStatus.PNSlaveNotOnline);

	    IF #iqUDT_VSUInterface.ResetStatistics OR #sUDT_HMIStatus.PNSlaveNotOnline
	    THEN

	        "FC_Statistics"(ix_Reset := #iqUDT_VSUInterface.ResetStatistics,
	                        ix_Activate := #sUDT_HMIStatus.PNSlaveNotOnline,
	                        ix_RTrigActivate := #sR_TRIG_PNSlaveNotOnline.Q,
	                        iqUDT_Statistics := #iqUDT_Statistics.PNSlaveNotOnline);
	    END_IF;

	    // create trigger on error and create statistics for profinet slave error
	    #sR_TRIG_PNSlaveError(CLK := #sUDT_HMIStatus.PNSlaveError);

	    IF #iqUDT_VSUInterface.ResetStatistics OR #sUDT_HMIStatus.PNSlaveError
	    THEN

	        "FC_Statistics"(ix_Reset := #iqUDT_VSUInterface.ResetStatistics,
	                        ix_Activate := #sUDT_HMIStatus.PNSlaveError,
	                        ix_RTrigActivate := #sR_TRIG_PNSlaveError.Q,
	                        iqUDT_Statistics := #iqUDT_Statistics.PNSlaveError);
	    END_IF;

	END_REGION

	REGION 7 - Status
	    // Statement section REGION
	    #iqUDT_VSUInterface.InternalErrorRIOPanel := #sUDT_HMIStatus.PNSlaveError
	    OR #sUDT_HMIStatus.PNSlaveNotOnline
	    OR #si_NrOfModulesWithError <> 0
	    OR #sUDT_HMIStatus."400VCircuitBreaker"
	    OR #sUDT_HMIStatus."24VPowersupplyError"
	    OR #sUDT_HMIStatus.BrakeCircuitBreaker
	    OR #sUDT_HMIStatus.BrakeThermalError;

	    // HMI status update

	    #qUDT_HMIStatus := #sUDT_HMIStatus;                       // Copy HMI status to output

	END_REGION

END_FUNCTION_BLOCK

FUNCTION_BLOCK "FB_Lift"
TITLE = FB_Lift
{ S7_Optimized_Access := 'TRUE' }
VERSION : 0.1
// ATTRIBUTES
// AUTO_NUMBER = True
// BLOCK_NUMBER = 198
// END_ATTRIBUTES
//Function to generate a position decision and handle conveyors around the in and outfeed of a lift
   VAR_INPUT
      iUDT_LiftConveyorInterface { ExternalAccessible := 'False'; ExternalVisible := 'False'; ExternalWritable := 'False'} : "UDT_ConveyorInterface";   // Interface structure
      iUDT_VSUInterface { ExternalAccessible := 'False'; ExternalVisible := 'False'; ExternalWritable := 'False'} : "UDT_VSUInterface";   // Interface between VSU and VFD
      ix_SectionIsDown { ExternalAccessible := 'False'; ExternalVisible := 'False'; ExternalWritable := 'False'} : Bool;   // TRUE when section is down
      ix_SectionIsUp { ExternalAccessible := 'False'; ExternalVisible := 'False'; ExternalWritable := 'False'} : Bool;   // TRUE when section is up
      ix_PECLift { ExternalAccessible := 'False'; ExternalVisible := 'False'; ExternalWritable := 'False'} : Bool;   // TRUE when PEC on lift is free
      ix_ConveyorEmptyInAuto { ExternalAccessible := 'False'; ExternalVisible := 'False'; ExternalWritable := 'False'} : Bool;   // Conveyor is started in auto
      ix_ConveyorEmptyOutAuto { ExternalAccessible := 'False'; ExternalVisible := 'False'; ExternalWritable := 'False'} : Bool;   // Conveyor is started in auto
      ix_ConveyorFullInAuto { ExternalAccessible := 'False'; ExternalVisible := 'False'; ExternalWritable := 'False'} : Bool;   // Conveyor is started in auto
      ix_ConveyorFullOutAuto { ExternalAccessible := 'False'; ExternalVisible := 'False'; ExternalWritable := 'False'} : Bool;   // Conveyor is started in auto
   END_VAR

   VAR_OUTPUT
      qi_RequestedPosition { ExternalAccessible := 'False'; ExternalVisible := 'False'; ExternalWritable := 'False'} : Int;   // Requested position to go to
      qx_HoldLiftConveyor { ExternalAccessible := 'False'; ExternalVisible := 'False'; ExternalWritable := 'False'} : Bool;   // Hold conveyor on lift as lift moves
      qx_TransportIdle { ExternalAccessible := 'False'; ExternalVisible := 'False'; ExternalWritable := 'False'} : Bool;   // No transports are active, free to move
      qx_LiftConveyorDirection { ExternalAccessible := 'False'; ExternalVisible := 'False'; ExternalWritable := 'False'} : Bool;   // FALSE - Right, TRUE - Left
   END_VAR

   VAR_IN_OUT
      iqUDT_LiftConveyorHandShakeUpstream : "UDT_ConveyorHandshake";
      iqUDT_LiftConveyorHandShake : "UDT_ConveyorHandshake";
      iqUDT_InfeedEmptyUpHandShake : "UDT_ConveyorHandshake";
      iqUDT_OutfeedEmptyDownHandShake : "UDT_ConveyorHandshake";
      iqUDT_InfeedFullDownHandShake : "UDT_ConveyorHandshake";
      iqUDT_OutfeedFullUpHandShake : "UDT_ConveyorHandshake";
      iqUDT_OutfeedFullUpHandshakeUpstream : "UDT_ConveyorHandshake";
      iqUDT_OutfeedEmptyDownHandshakeUpstream : "UDT_ConveyorHandshake";
   END_VAR

